INTERFACE PUBLIC MoveBuilder EXTENDS __System.IQueryInterface

METHOD PUBLIC Acceleration : MoveBuilder
VAR_INPUT
	value : LREAL;
END_VAR
END_METHOD

METHOD PUBLIC BufferMode : MoveBuilder
VAR_INPUT
	mode : MotionBufferMode;
END_VAR
END_METHOD

METHOD PUBLIC BuildMoveVelocityCommand : MoveCommand
VAR_INPUT
	axis : REFERENCE TO Mc2Axis;
END_VAR
END_METHOD

METHOD PUBLIC Deceleration : MoveBuilder
VAR_INPUT
	value : LREAL;
END_VAR
END_METHOD

METHOD PUBLIC Distance : MoveRelativeBuilder
VAR_INPUT
	value : LREAL;
END_VAR
END_METHOD

METHOD PUBLIC Jerk : MoveBuilder
VAR_INPUT
	value : LREAL;
END_VAR
END_METHOD

METHOD PUBLIC Position : MoveAbsoluteBuilder
VAR_INPUT
	value : LREAL;
END_VAR
END_METHOD

METHOD PUBLIC Reset : MoveBuilder
END_METHOD

METHOD PUBLIC Velocity : MoveBuilder
VAR_INPUT
	value : LREAL;
END_VAR
END_METHOD

END_INTERFACE

(* stored: Version 1.1.0.1
   Itf MoveBuilder: Id {2515b8d1-881d-0ccb-15a6-7d04a4e73429}
   Method Acceleration: Id {a50d0b42-c60e-06d2-0dc7-a428b5bd2858}
   Method BufferMode: Id {8058df80-7c06-0a07-018e-a453bfa23e97}
   Method BuildMoveVelocityCommand: Id {0fd3c392-d1e2-06f3-2fa5-d8869d117ef5}
   Method Deceleration: Id {4f849c2b-2837-0ef6-3983-b8af5bf49e80}
   Method Distance: Id {ccf28c55-362b-01fc-3ee6-b57b36715a07}
   Method Jerk: Id {ff2bdc64-e58b-0579-3e8d-dece01005d36}
   Method Position: Id {062b27ce-68c0-01a3-03b0-70dfca1efac6}
   Method Reset: Id {84b0d7e3-ce89-06b9-389b-7164012f5ce1}
   Method Velocity: Id {9b858d16-c130-0881-30d5-ac32592effd9} *)
